FUNCTION_BLOCK DoseInit EXTENDS BaseState
VAR_INPUT
END_VAR
VAR_OUTPUT
END_VAR
VAR
END_VAR

METHOD mIrun : BOOL
FOR Index:=1 TO BasePointer^.pNUM_SILOS BY 1 DO
	IF BasePointer^.LoadCellOutput[INDEX].ScaledValue < BasePointer^.SiloFlagsAccessI[INDEX].pTargetWeight THEN
		BasePointer^.SiloFlagsAccessI[INDEX].pLowProduct := TRUE;	
	ELSE
		BasePointer^.SiloFlagsAccessI[INDEX].pLowProduct := FALSE;
	END_IF
		
	BasePointer^.SiloFlagsAccessI[Index].pBufferedWeight := BasePointer^.LoadCellOutput[Index].ScaledValue;
	BasePointer^.SpiralAccessI[Index].mAutoOn();
	BasePointer^.MachineFlagsAccessI.pDosing := TRUE;
END_FOR

mNextState();
END_METHOD

END_FUNCTION_BLOCK

(* stored: Version 1.1.0.1, ProductVersion 3.1.4024.12
   POU DoseInit: Id {f3b157e4-48d9-48be-885b-a12cb1b2f9b1}, SpecialFunc None
   Method mIrun: Id {29849357-84d1-471f-87ca-bd7248ba737d} *)
